Staubli VAL3: TrajPointItem.dtx

public TrajectoryItem tSuper
  [0]
    num distance
    num moveType
    num nTime
    num nStop
    num nTcpAction
    string comment
    bool toStop
    mdesc nom_speed = {vel=450, tmax=1000}
    InstrItem iInstr[3]
      [0]
        string sType
        string sData
      [1]
        string sType
        string sData
      [2]
        string sType
        string sData
    num nMoveId
public pointRx pPoint = {fatherId=world[0]}
public num nType
